(*
Will be an abstract class that will be used to configure all parts of the machine through json
*)

FUNCTION_BLOCK ABSTRACT FB_ConfigJson
VAR_INPUT
END_VAR
VAR_OUTPUT
END_VAR
VAR 
	_fbName : STRING; //name of FB set on init
END_VAR

METHOD _F_Axis : HRESULT
VAR_IN_OUT
	a_pstAxisParameterSet : POINTER TO Tc2_MC2.ST_AxisParameterSet; //pointer to array
	pstAxisMapping : UDINT;
END_VAR
END_METHOD

METHOD PROTECTED ABSTRACT _F_IO : HResult
VAR_IN_OUT
	a_pstIOMappingJson : POINTER TO ST_IOMappingJson; //pointer to array
	ustIOMappingJson : UDINT; 		
END_VAR
END_METHOD

(*
return the list of vars that want to be saved and loaded 
*)

METHOD PROTECTED ABSTRACT _F_Recipe : HResult
VAR_IN_OUT
	a_pstAnyTypeUser : POINTER TO MPM_JsonParser.ST_AnyType_User; //pointer to array
	uAnyTypeUser : UDINT; //size of array	
END_VAR
VAR_OUTPUT

END_VAR
END_METHOD

METHOD PROTECTED ABSTRACT _F_System : HResult
VAR_IN_OUT
	a_pstAnyTypeUser : POINTER TO MPM_JsonParser.ST_AnyType_User; //pointer to array
	uAnyTypeUser : UDINT; //size of array	
END_VAR
END_METHOD

METHOD PUBLIC FINAL F_AXIS : HRESULT
VAR_INPUT
	lastResult : HRESULT;
	sJson : SJsonValue;
	pfbJsonSchema : POINTER TO FB_NCAxisJson_V2;	
	bGet : BOOL;
END_VAR

VAR_INST
	_fbResult : FB_ResultHelper_V2;
	pResult : POINTER TO HRESULT;
END_VAR

VAR
	a_pstAxisParameterSet : POINTER TO Tc2_MC2.ST_AxisParameterSet;
	dstAxisParameterSet : UDINT; //number of bytes in a_stAnyUser
	
	uSizeOfArray : UDINT;
	
	pstAxisParameterSet : POINTER TO Tc2_MC2.ST_AxisParameterSet; //pointer for loop
	x : UDINT;
END_VAR


VAR CONSTANT
	uSizeOfStAnyType : UDINT := SIZEOF(Tc2_MC2.ST_AxisParameterSet);
END_VAR
IF _fbResult.M_MethodResult(F_AXIS,ADR(pResult),lastResult) = FALSE THEN
	RETURN;
END_IF


pResult^ := _F_Axis(a_pstAxisParameterSet,dstAxisParameterSet);
//pResult^ := MPM_FBResult.E_Result.S_WORKING;
IF bGet = FALSE THEN
	sJson := pfbJsonSchema^.M_SetJsonMember(sJson,_fbName);
	IF a_pstAxisParameterSet > 0 AND dstAxisParameterSet > 0 AND uSizeOfStAnyType > 0 THEN //make sure all values are vaild
		uSizeOfArray := dstAxisParameterSet/uSizeOfStAnyType - 1; //get number of items in array
		FOR x := 0 TO uSizeOfArray BY 1 DO //loop through all items 
			pstAxisParameterSet := a_pstAxisParameterSet + uSizeOfStAnyType*x; // get array position
			pResult^ := pfbJsonSchema^.M_SetAxisJson(pResult^,sJson,pstAxisParameterSet);
		END_FOR
	END_IF	
ELSIF bGet = TRUE THEN
	sJson := pfbJsonSchema^.FindMember(sJson,_fbName);
	IF a_pstAxisParameterSet > 0 AND dstAxisParameterSet > 0 AND uSizeOfStAnyType > 0 THEN //make sure all values are vaild
		uSizeOfArray := dstAxisParameterSet/uSizeOfStAnyType - 1; //get number of items in array
		FOR x := 0 TO uSizeOfArray BY 1 DO //loop through all items 
			pstAxisParameterSet := a_pstAxisParameterSet + uSizeOfStAnyType*x; // get array position
			pResult^ := pfbJsonSchema^.M_GetAxisJson(pResult^,sJson,pstAxisParameterSet);
		END_FOR
	END_IF
END_IF
END_METHOD

METHOD PUBLIC FINAL F_IO : HRESULT
VAR_INPUT
	lastResult : HRESULT;
	sJson : SJsonValue;
	pfbJsonSchema : POINTER TO FB_JsonSchemaEx_OLD;
	bGet : BOOL;	
END_VAR

VAR_INST
	_fbResult : FB_ResultHelper_V2;
	pResult : POINTER TO HRESULT;
END_VAR

VAR
	a_pstIOMappingJson : POINTER TO ST_IOMappingJson; // pointer to array of vars
	uAnyTypeUser : UDINT; //number of bytes in a_stAnyUser
	
	uSizeOfArray : UDINT;
	pstIOMappingJson : POINTER TO ST_IOMappingJson; //pointer for loop
	x : UDINT;
END_VAR


VAR CONSTANT
	uSizeOfStAnyType : UDINT := SIZEOF(ST_IOMappingJson);
END_VAR
IF _fbResult.M_MethodResult(F_IO,ADR(pResult),lastResult) = FALSE THEN
	RETURN;
END_IF


pResult^ := _F_IO(a_pstIOMappingJson,uAnyTypeUser); //gets pointer from FB


pResult^ := MPM_FBResult.E_Result.S_WORKING;
//set
IF bGet = FALSE THEN
	sJson := pfbJsonSchema^.M_SetJsonMember(sJson,_fbName);
	IF a_pstIOMappingJson > 0 AND_THEN uAnyTypeUser > 0 AND uSizeOfStAnyType > 0 THEN //make sure all values are vaild
		uSizeOfArray := uAnyTypeUser/uSizeOfStAnyType - 1; //get number of items in array
		FOR x := 0 TO uSizeOfArray BY 1 DO //loop through all items 
			pstIOMappingJson := a_pstIOMappingJson + uSizeOfStAnyType*x; // get array position
			sJson := pfbJsonSchema^.M_SetJsonMember(sJson,pstIOMappingJson^.name); //set json value
			pfbJsonSchema^.M_SetJsonMemberValue(sJson,'channel',pstIOMappingJson^.channel); //set json value
			pfbJsonSchema^.M_SetJsonMemberValue(sJson,'deviceNum',pstIOMappingJson^.deviceNum); //set json value
			pfbJsonSchema^.M_SetJsonMemberValue(sJson,'ethercatDeviceNum',pstIOMappingJson^.ethercatDeviceNum); //set json value
			pfbJsonSchema^.M_SetJsonMemberValue(sJson,'ioLinkDevice',pstIOMappingJson^.ioLinkDevice); //set json value
			pfbJsonSchema^.M_SetJsonMemberValue(sJson,'ioLinkSlaveChannel',pstIOMappingJson^.ioLinkSlaveChannel); //set json value
		END_FOR
		pResult^ := MPM_FBResult.E_Result.S_OK;
	ELSE
		pResult^ := MPM_FBResult.E_Result.S_FAILED;
	END_IF
//get
ELSIF bGet = TRUE THEN
	sJson := pfbJsonSchema^.FindMember(sJson,_fbName);
	IF a_pstIOMappingJson > 0 AND_THEN uAnyTypeUser > 0 AND uSizeOfStAnyType > 0 THEN //make sure all values are vaild
		uSizeOfArray := uAnyTypeUser/uSizeOfStAnyType - 1; //get number of items in array
		FOR x := 0 TO uSizeOfArray BY 1 DO //loop through all items 
			pstIOMappingJson := a_pstIOMappingJson + uSizeOfStAnyType*x; // get array position
			sJson := pfbJsonSchema^.M_SetJsonMember(sJson,pstIOMappingJson^.name); //set json value
			pfbJsonSchema^.M_GetJsonMemberValue(sJson,'channel',pstIOMappingJson^.channel); //set json value
			pfbJsonSchema^.M_GetJsonMemberValue(sJson,'deviceNum',pstIOMappingJson^.deviceNum); //set json value
			pfbJsonSchema^.M_GetJsonMemberValue(sJson,'ethercatDeviceNum',pstIOMappingJson^.ethercatDeviceNum); //set json value
			pfbJsonSchema^.M_GetJsonMemberValue(sJson,'ioLinkDevice',pstIOMappingJson^.ioLinkDevice); //set json value
			pfbJsonSchema^.M_GetJsonMemberValue(sJson,'ioLinkSlaveChannel',pstIOMappingJson^.ioLinkSlaveChannel); //set json value
		END_FOR
		pResult^ := MPM_FBResult.E_Result.S_OK;
	ELSE
		pResult^ := MPM_FBResult.E_Result.S_FAILED;
	END_IF
END_IF
END_METHOD

METHOD PROTECTED F_Map_ST_IOMappingJson : HRESULT
VAR_INPUT
	stIOMappingJson : POINTER TO ST_IOMappingJson;
	name : STRING;
	pPVoid : POINTER TO PVOID;
END_VAR
END_METHOD

METHOD PUBLIC FINAL F_Recipe : HRESULT
VAR_INPUT
	lastResult : HRESULT;
	sJson : SJsonValue;
	pfbJsonSchema : POINTER TO FB_JsonSchemaEx_OLD;	
	bGet : BOOL;
END_VAR

VAR_INST
	_fbResult : FB_ResultHelper_V2;
	pResult : POINTER TO HRESULT;
END_VAR

VAR
	a_stAnyUser : POINTER TO MPM_JsonParser.ST_AnyType_User; // pointer to array of vars
	uAnyTypeUser : UDINT; //number of bytes in a_stAnyUser
	
	uSizeOfArray : UDINT;
	pstAnyUser : POINTER TO MPM_JsonParser.ST_AnyType_User; //pointer for loop
	x : UDINT;
END_VAR

VAR CONSTANT
	uSizeOfStAnyType : UDINT := SIZEOF(MPM_JsonParser.ST_AnyType_User);
END_VAR
IF _fbResult.M_MethodResult(F_Recipe,ADR(pResult),lastResult) = FALSE THEN
	RETURN;
END_IF


pResult^ := _F_Recipe(a_stAnyUser,uAnyTypeUser);


pResult^ := MPM_FBResult.E_Result.S_WORKING;

//set
IF bGet = FALSE THEN
	sJson := pfbJsonSchema^.M_SetJsonMember(sJson,_fbName);
	IF a_stAnyUser > 0 AND_THEN uAnyTypeUser > 0 AND uSizeOfStAnyType > 0 THEN //make sure all values are vaild
		uSizeOfArray := uAnyTypeUser/uSizeOfStAnyType - 1; //get number of items in array
		FOR x := 0 TO uSizeOfArray BY 1 DO //loop through all items 
			pstAnyUser := a_stAnyUser + uSizeOfStAnyType*x; // get array position
				pfbJsonSchema^.M_SetJsonMemberValue_AnyType(sJson,pstAnyUser^.name,pstAnyUser^); //set json value
		END_FOR
		pResult^ := MPM_FBResult.E_Result.S_OK;
	ELSE
		pResult^ := MPM_FBResult.E_Result.S_FAILED;
	END_IF
	
//get
ELSIF bGet = TRUE THEN 	
	sJson := pfbJsonSchema^.FindMember(sJson,_fbName);
	IF a_stAnyUser > 0 AND_THEN uAnyTypeUser > 0 AND uSizeOfStAnyType > 0 THEN //make sure all values are vaild
		uSizeOfArray := uAnyTypeUser/uSizeOfStAnyType - 1; //get number of items in array
		FOR x := 0 TO uSizeOfArray BY 1 DO //loop through all items 
			pstAnyUser := a_stAnyUser + uSizeOfStAnyType*x; // get array position
				pfbJsonSchema^.M_GetJsonMemberValue_AnyType(sJson,pstAnyUser^.name,pstAnyUser^); //set json value
		END_FOR
		pResult^ := MPM_FBResult.E_Result.S_OK;
	ELSE
		pResult^ := MPM_FBResult.E_Result.S_FAILED;
	END_IF
END_IF
END_METHOD

METHOD PUBLIC FINAL F_System : HRESULT
VAR_INPUT
	lastResult : HRESULT;
	sJson : SJsonValue;
	pfbJsonSchema : POINTER TO FB_JsonSchemaEx_OLD;	
	bGet : BOOL;	
END_VAR

VAR_INST
	_fbResult : FB_ResultHelper_V2;
	pResult : POINTER TO HRESULT;
END_VAR

VAR
	a_stAnyUser : POINTER TO MPM_JsonParser.ST_AnyType_User; // pointer to array of vars
	uAnyTypeUser : UDINT; //number of bytes in a_stAnyUser
	
	uSizeOfArray : UDINT;
	pstAnyUser : POINTER TO MPM_JsonParser.ST_AnyType_User; //pointer for loop
	x : UDINT;
END_VAR


VAR CONSTANT
	uSizeOfStAnyType : UDINT := SIZEOF(MPM_JsonParser.ST_AnyType_User);
END_VAR
IF _fbResult.M_MethodResult(F_System,ADR(pResult),lastResult) = FALSE THEN
	RETURN;
END_IF


pResult^ := _F_System(a_stAnyUser,uAnyTypeUser);
//set
IF bGet = FALSE THEN
	pResult^ := MPM_FBResult.E_Result.S_WORKING;
	sJson := pfbJsonSchema^.M_SetJsonMember(sJson,_fbName);
	IF a_stAnyUser > 0 AND_THEN uAnyTypeUser > 0 AND uSizeOfStAnyType > 0 THEN //make sure all values are vaild
		uSizeOfArray := uAnyTypeUser/uSizeOfStAnyType - 1; //get number of items in array
		FOR x := 0 TO uSizeOfArray BY 1 DO //loop through all items 
			pstAnyUser := a_stAnyUser + uSizeOfStAnyType*x; // get array position
				pfbJsonSchema^.M_SetJsonMemberValue_AnyType(sJson,pstAnyUser^.name,pstAnyUser^); //set json value
		END_FOR
		pResult^ := MPM_FBResult.E_Result.S_OK;
	ELSE
		pResult^ := MPM_FBResult.E_Result.S_FAILED;
	END_IF

//get	
ELSIF bGet = TRUE THEN
	sJson := pfbJsonSchema^.FindMember(sJson,_fbName);
	IF a_stAnyUser > 0 AND_THEN uAnyTypeUser > 0 AND uSizeOfStAnyType > 0 THEN //make sure all values are vaild
		uSizeOfArray := uAnyTypeUser/uSizeOfStAnyType - 1; //get number of items in array
		FOR x := 0 TO uSizeOfArray BY 1 DO //loop through all items 
			pstAnyUser := a_stAnyUser + uSizeOfStAnyType*x; // get array position
				pfbJsonSchema^.M_GetJsonMemberValue_AnyType(sJson,pstAnyUser^.name,pstAnyUser^); //set json value
		END_FOR
		pResult^ := MPM_FBResult.E_Result.S_OK;
	ELSE
		pResult^ := MPM_FBResult.E_Result.S_FAILED;
	END_IF	
END_IF
END_METHOD

METHOD FB_init : BOOL
VAR_INPUT
	bInitRetains : BOOL; // if TRUE, the retain variables are initialized (warm start / cold start)
	bInCopyCode : BOOL;  // if TRUE, the instance afterwards gets moved into the copy code (online change)
	fbName : STRING;
END_VAR
_fbName := fbName;
END_METHOD

PROPERTY PUBLIC P_fbName : STRING
GET
P_fbName := _fbName;
END_GET
END_PROPERTY

END_FUNCTION_BLOCK

(* stored: Version 1.1.0.1, ProductVersion 3.1.4024.12
   POU FB_ConfigJson: Id {3ccc0d41-27f9-41ab-b33f-1e963a615b44}, SpecialFunc None
   Folder ABSTRACT: Id {d3f0e259-1061-426a-b7a1-3591a9d5be2f}
   Folder Protected: Id {d31bea82-4c8d-4864-8213-7cfbba3c0754}
   Method _F_Axis: Id {7fa39416-568e-4119-8393-652fc6472acb}
   Method _F_IO: Id {25f7451c-b2be-4782-91c3-53451c901d29}
   Method _F_Recipe: Id {acb8c5d6-5487-4d41-9ec0-f4a34dd65731}
   Method _F_System: Id {c67585fa-6db9-4ba3-8b65-2665a130374f}
   Method F_AXIS: Id {c0243cb9-9b32-4370-9384-0993220a2226}
   Method F_IO: Id {3a02837e-fabe-4f90-b88e-c4f1e99bdab4}
   Method F_Map_ST_IOMappingJson: Id {5c1ae8e3-b5c1-4247-821a-ef4678ae72df}
   Method F_Recipe: Id {23f9deca-2586-4a9d-b0ee-68078bcc9c57}
   Method F_System: Id {4f92d8d9-026e-4619-8a71-a0cfc6eb2eed}
   Method FB_init: Id {39c76da8-be3f-4311-946f-56a7e0460487}
   Property P_fbName: Id {5a2b393b-8b77-4ed7-a71a-7e64119bd062}
   Get Get: Id {831f96df-87bd-4bb9-ad06-74017936567e} *)
